# EPICS autosave request: iocBoot/sioc-in10-im02/sioc-in10-im02.req
file "facet2.req" AREA=IN10,POS=791
file "facet2.req" AREA=LI11,POS=360
